TYPE (* A Subrange Data Type *)
  (* Standard: 61131-3 *)
  (* Version 0.0, 2003-12-06, JHC, Rockwell Automation *)
  (* Compiler header: package fb.rt.template; *)
  (* Compiler Java IBM VisualAge 3.0 *)
  (* ASN.1 tag PRIVATE 9 *)
  Subrange : INT(-4095..4095);
END_TYPE
